TYPE "UDT_TrackingReport_HMI_OP1_ext"
VERSION : 0.1
   STRUCT
      ClearReport : Bool;
      PosInx_HMI : Int;
      PageNo : Int;
      RowIndex : Array[0..9] of Int;
   END_STRUCT;

END_TYPE

